// TIA Portal project "siemens_tia19" (V19)

(* hardware
DEVICE "S71500/ET200MP station_1"  S7-1500 station
   slot 0: "Rail_0"  Rack  6ES7 590-1***0-0AA0
   slot 1: "PLC_1"  CPU 1515-2 PN  6ES7 515-2AM02-0AB0  V2.8
      slot 3: "CPU display_1"  6ES7591-1BA00-0AA0
      slot 32768: "PROFINET interface_1"  X1
         slot 32769: "Port_1"  X1 P1
         slot 32770: "Port_2"  X1 P2
      slot 33024: "PROFINET interface_2"  X2
         slot 33025: "Port_1"  X2 P1
      slot 34817: "Virtual CP interface port_1"  Virtual CP interface port  Virtual CP interface port
DEVICE "ET 200SP station_1"  ET 200SP-Station
   slot 0: "Rack_0"  Rack  6ES5 710-8MAx1
   slot 0: "IO device_1"  IM 155-6 PN ST  6ES7 155-6AU00-0BN0  V3.3
   slot 1: "DI 8x24VDC HF_1"  DI 8x24VDC HF  6ES7 131-6BF00-0CA0  V1.2
      slot 1: "DI 8x24VDC HF_1"  DI 8x24VDC HF
   slot 2: "DI 8x24VDC HF_2"  DI 8x24VDC HF  6ES7 131-6BF00-0CA0  V1.2
      slot 1: "DI 8x24VDC HF_2"  DI 8x24VDC HF
   slot 3: "AI 4xU/I 2-wire ST_1"  AI 4xU/I 2-wire ST  6ES7 134-6HD01-0BA1  V2.0
      slot 1: "AI 4xU/I 2-wire ST_1"  AI 4xU/I 2-wire ST
   slot 4: "Server module_1"  Server module  6ES7 193-6PA00-0AA0  V1.1
      slot 1: "Server module_1"  Server module
   slot 127: "BA 2xRJ45"  BA 2xRJ45  6ES7 193-6AR00-0AA0  V0.0
      slot 1: "Port_1"  X1 P1 R  6ES7 193-6AR00-0AA0  V0.0
      slot 2: "Port_2"  X1 P2 R  6ES7 193-6AR00-0AA0  V0.0
*)

// ===== PLC "PLC_1"  CPU 1515-2 PN =====

VAR_GLOBAL   // PLC tag table "Default tag table"
   "DI_0" AT %I0.0 : Bool;
   "DI_1" AT %I0.1 : Bool;
   "DI_2" AT %I0.2 : Bool;
   "DI_3" AT %I0.3 : Bool;
   "DI_4" AT %I0.4 : Bool;
   "DI_5" AT %I0.5 : Bool;
   "DI_6" AT %I0.6 : Bool;
   "DI_7" AT %I0.7 : Bool;
   "DI_8" AT %I1.0 : Bool;
   "DI_9" AT %I1.1 : Bool;
   "DI_10" AT %I1.2 : Bool;
   "DI_11" AT %I1.3 : Bool;
   "DI_12" AT %I1.4 : Bool;
   "DI_13" AT %I1.5 : Bool;
   "DI_14" AT %I1.6 : Bool;
   "DI_15" AT %I1.7 : Bool;
   "AI_1" AT %IW2 : Int;
   "AI_2" AT %IW4 : Int;
   "AI_3" AT %IW6 : Int;
   "AI_4" AT %IW8 : Int;
   "Clock_Byte" AT %MB0 : Byte;
   "Clock_10Hz" AT %M0.0 : Bool;
   "Clock_5Hz" AT %M0.1 : Bool;
   "Clock_2.5Hz" AT %M0.2 : Bool;
   "Clock_2Hz" AT %M0.3 : Bool;
   "Clock_1.25Hz" AT %M0.4 : Bool;
   "Clock_1Hz" AT %M0.5 : Bool;
   "Clock_0.625Hz" AT %M0.6 : Bool;
   "Clock_0.5Hz" AT %M0.7 : Bool;
END_VAR

DATA_BLOCK "DB_ET200SP"   // DB1
{ S7_Optimized_Access := 'TRUE' }
VERSION : 0.1
   VAR
      Output1 : Bool;   // Hello, World!
      Output2 : Bool;
      "Timer" : TON_TIME;
      AI_1_V : Real;
      AI_2_V : Real;
      AI_3_V : Real;
      AI_4_V : Real;
   END_VAR
BEGIN
END_DATA_BLOCK

DATA_BLOCK "ConvertAnalogRawToReal_DB"   // DB2
{ S7_Optimized_Access := 'TRUE' }
VERSION : 0.1
// stored: InstanceOfName ConvertAnalogRawToReal
"ConvertAnalogRawToReal"
BEGIN
END_DATA_BLOCK

FUNCTION_BLOCK "ConvertAnalogRawToReal"   // FB1, SCL
{ S7_Optimized_Access := 'TRUE' }
VERSION : 0.1
   VAR_INPUT
      AnalogRaw : Int;
   END_VAR
   VAR_OUTPUT
      AnalogReal : Real;
   END_VAR
   VAR CONSTANT
      MIN_VOLTAGE_RAW : Real := -29038.0;
      MAX_VOLTAGE_RAW : Real := 29007.0;
      MIN_VOLTAGE_REAL : Real := -10.38;
      MAX_VOLTAGE_REAL : Real := 10.38;
   END_VAR
BEGIN
   #AnalogReal := (#AnalogRaw - #MIN_VOLTAGE_RAW) / (#MAX_VOLTAGE_RAW - #MIN_VOLTAGE_RAW) * (#MAX_VOLTAGE_REAL - #MIN_VOLTAGE_REAL) + #MIN_VOLTAGE_REAL;
END_FUNCTION_BLOCK

ORGANIZATION_BLOCK "Main"   // OB1, SCL, ProgramCycle
TITLE = "Main Program Sweep (Cycle)"
{ S7_Optimized_Access := 'TRUE' }
VERSION : 0.1
   VAR_INPUT
      Initial_Call : Bool;   // Initial call of this OB
      Remanence : Bool;   // =True, if remanent data are available
   END_VAR
   VAR CONSTANT
      MIN_VOLTAGE_RAW : Real := -29038.0;
      MAX_VOLTAGE_RAW : Real := 29007.0;
      MIN_VOLTAGE_REAL : Real := -10.38;
      MAX_VOLTAGE_REAL : Real := 10.38;
   END_VAR
BEGIN
   IF "DB_ET200SP".Output1 THEN
     "DB_ET200SP".Output1 := "DI_0";
   END_IF;


   "DB_ET200SP".Output1 := "Clock_10Hz";

   "DB_ET200SP".Timer(IN := "DI_0",
                      PT := T#3S);
   "DB_ET200SP".Output2 := "DB_ET200SP".Timer.Q;

   // Convert Analog Inputs to Voltage (as real)
   "ConvertAnalogRawToReal_DB"(AnalogRaw:="AI_1",
                               AnalogReal=>"DB_ET200SP".AI_1_V);
   "ConvertAnalogRawToReal_DB"(AnalogRaw := "AI_2",
                               AnalogReal => "DB_ET200SP".AI_2_V);
   "ConvertAnalogRawToReal_DB"(AnalogRaw := "AI_3",
                               AnalogReal => "DB_ET200SP".AI_3_V);
   "ConvertAnalogRawToReal_DB"(AnalogRaw := "AI_4",
                               AnalogReal => "DB_ET200SP".AI_4_V);
END_ORGANIZATION_BLOCK